{attribute 'qualified_only'}
{attribute 'strict'}
TYPE E_PIZZA_TYPES :
(
	eType_Cheese := 0,
	eType_Pepperoni := 1,
	eType_Olives := 2
);
END_TYPE

(* stored: Version 1.1.0.1, ProductVersion 3.1.4024.12
   DUT E_PIZZA_TYPES: Id {ce81d71e-5d40-4b85-b465-119161746432} *)
